PROGRAM Presseurs_Laser
VAR
FB_Presseurs_K11_Amont_Laser, 
FB_Presseurs_L12_Aval_Laser	: FB_Presseurs_LASER;

	Test_Serr,	test_Desser,Test_Serr2,	test_Desser2	:BOOL;


END_VAR

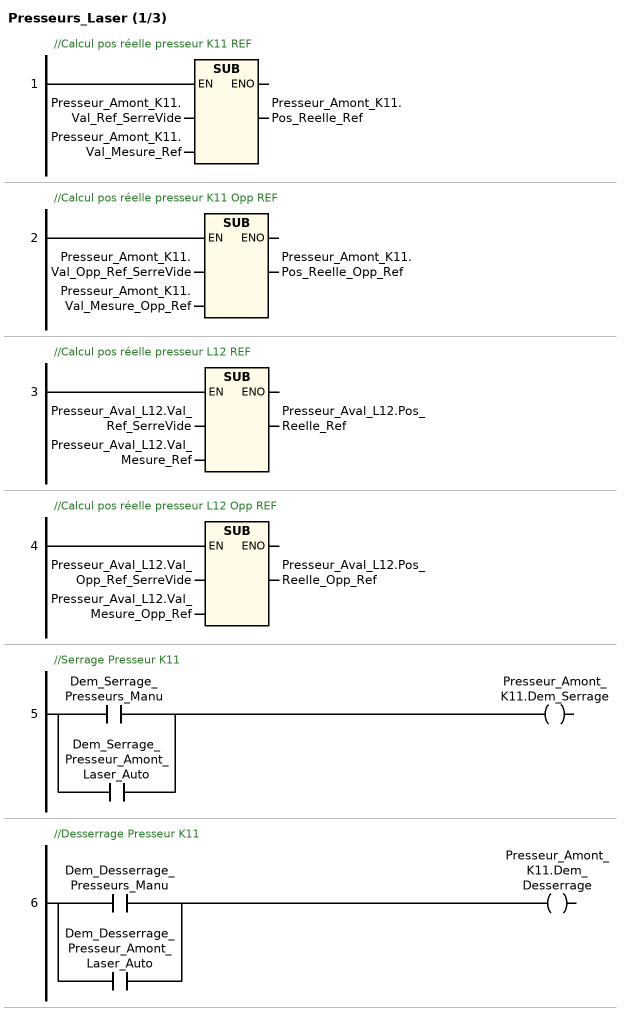
// NETWORK 1
// //Calcul pos réelle presseur K11 REF
Presseur_Amont_K11.Pos_Reelle_Ref := Presseur_Amont_K11.Val_Ref_SerreVide - Presseur_Amont_K11.Val_Mesure_Ref;

// NETWORK 2
// //Calcul pos réelle presseur K11 Opp REF
Presseur_Amont_K11.Pos_Reelle_Opp_Ref := Presseur_Amont_K11.Val_Opp_Ref_SerreVide - Presseur_Amont_K11.Val_Mesure_Opp_Ref;

// NETWORK 3
// //Calcul pos réelle presseur L12 REF
Presseur_Aval_L12.Pos_Reelle_Ref := Presseur_Aval_L12.Val_Ref_SerreVide - Presseur_Aval_L12.Val_Mesure_Ref;

// NETWORK 4
// //Calcul pos réelle presseur L12 Opp REF
Presseur_Aval_L12.Pos_Reelle_Opp_Ref := Presseur_Aval_L12.Val_Opp_Ref_SerreVide - Presseur_Aval_L12.Val_Mesure_Opp_Ref;

// NETWORK 5
// //Serrage Presseur K11
Presseur_Amont_K11.Dem_Serrage := Dem_Serrage_Presseurs_Manu OR Dem_Serrage_Presseur_Amont_Laser_Auto;

// NETWORK 6
// //Desserrage Presseur K11
Presseur_Amont_K11.Dem_Desserrage := Dem_Desserrage_Presseurs_Manu OR Dem_Desserrage_Presseur_Amont_Laser_Auto;

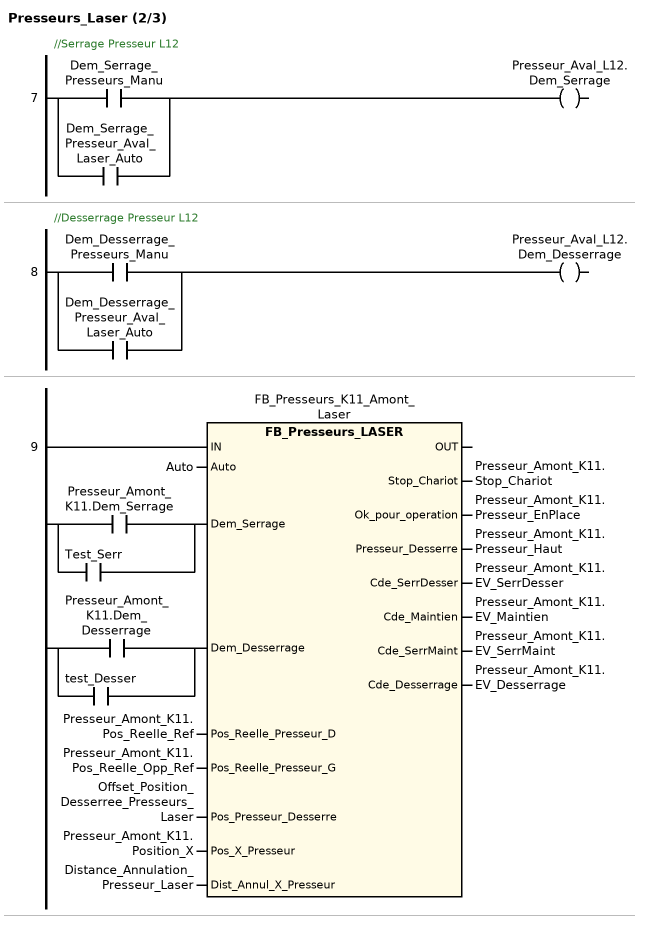
// NETWORK 7
// //Serrage Presseur L12
Presseur_Aval_L12.Dem_Serrage := Dem_Serrage_Presseurs_Manu OR Dem_Serrage_Presseur_Aval_Laser_Auto;

// NETWORK 8
// //Desserrage Presseur L12
Presseur_Aval_L12.Dem_Desserrage := Dem_Desserrage_Presseurs_Manu OR Dem_Desserrage_Presseur_Aval_Laser_Auto;

// NETWORK 9
FB_Presseurs_K11_Amont_Laser(
    IN := TRUE,
    Auto := Auto,
    Dem_Serrage := Presseur_Amont_K11.Dem_Serrage OR Test_Serr,
    Dem_Desserrage := Presseur_Amont_K11.Dem_Desserrage OR test_Desser,
    Pos_Reelle_Presseur_D := Presseur_Amont_K11.Pos_Reelle_Ref,
    Pos_Reelle_Presseur_G := Presseur_Amont_K11.Pos_Reelle_Opp_Ref,
    Pos_Presseur_Desserre := Offset_Position_Desserree_Presseurs_Laser,
    Pos_X_Presseur := Presseur_Amont_K11.Position_X,
    Dist_Annul_X_Presseur := Distance_Annulation_Presseur_Laser,
    Stop_Chariot => Presseur_Amont_K11.Stop_Chariot,
    Ok_pour_operation => Presseur_Amont_K11.Presseur_EnPlace,
    Presseur_Desserre => Presseur_Amont_K11.Presseur_Haut,
    Cde_SerrDesser => Presseur_Amont_K11.EV_SerrDesser,
    Cde_Maintien => Presseur_Amont_K11.EV_Maintien,
    Cde_SerrMaint => Presseur_Amont_K11.EV_SerrMaint,
    Cde_Desserrage => Presseur_Amont_K11.EV_Desserrage); // FB_Presseurs_LASER

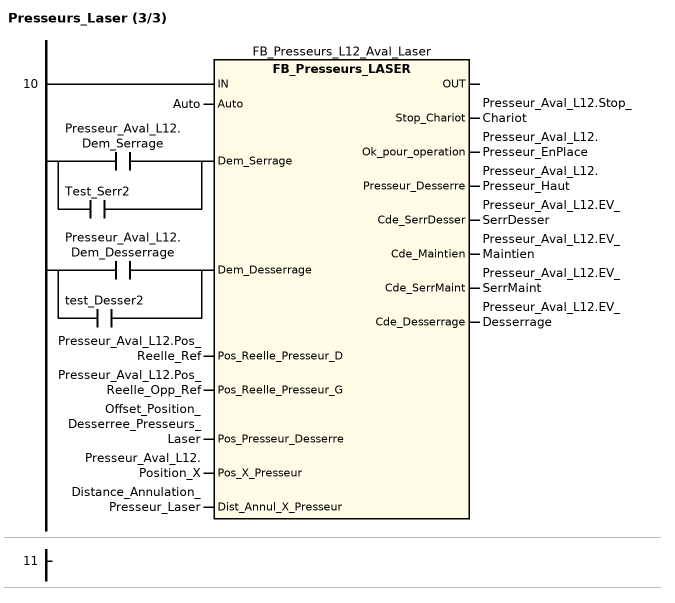
// NETWORK 10
FB_Presseurs_L12_Aval_Laser(
    IN := TRUE,
    Auto := Auto,
    Dem_Serrage := Presseur_Aval_L12.Dem_Serrage OR Test_Serr2,
    Dem_Desserrage := Presseur_Aval_L12.Dem_Desserrage OR test_Desser2,
    Pos_Reelle_Presseur_D := Presseur_Aval_L12.Pos_Reelle_Ref,
    Pos_Reelle_Presseur_G := Presseur_Aval_L12.Pos_Reelle_Opp_Ref,
    Pos_Presseur_Desserre := Offset_Position_Desserree_Presseurs_Laser,
    Pos_X_Presseur := Presseur_Aval_L12.Position_X,
    Dist_Annul_X_Presseur := Distance_Annulation_Presseur_Laser,
    Stop_Chariot => Presseur_Aval_L12.Stop_Chariot,
    Ok_pour_operation => Presseur_Aval_L12.Presseur_EnPlace,
    Presseur_Desserre => Presseur_Aval_L12.Presseur_Haut,
    Cde_SerrDesser => Presseur_Aval_L12.EV_SerrDesser,
    Cde_Maintien => Presseur_Aval_L12.EV_Maintien,
    Cde_SerrMaint => Presseur_Aval_L12.EV_SerrMaint,
    Cde_Desserrage => Presseur_Aval_L12.EV_Desserrage); // FB_Presseurs_LASER

// NETWORK 11

END_PROGRAM

(* stored: Version 1.1.0.1
   POU Presseurs_Laser: Id {4725ad0d-c44b-4c22-8b94-98ddfc1aad32}, SpecialFunc None *)
